VAR_GLOBAL
END_VAR

(* stored: Version 1.1.0.1, ProductVersion 3.1.4020.6
   GVL GVL_IO: Id {7514927d-6cd3-49a3-af7e-4b1a6475c939} *)
